(* Logix 5000 project; controller cal1632 1756-L62 rev 16.20; software revision 16.05; part 33 of 57 *)
(* tags used below, declared in another part *)
   FAULT : BOOL;
   HMI : BOOL;
   p01r03_lc3_ave_ctrl : CONTROL;
   p01r09_pb_global_reset : BOOL;
   p01r09_stretch_mode : BOOL;
   p02_real_from_hmi : hmi_real;
   p22_ai_amps : REAL;
   p22_ai_hz : REAL;
   p22_ai_speed : REAL;
   p22_ai_ts1_lc : REAL;
   p22_ao_selected_speed : REAL;
   p22_ao_torque : REAL;
   p22_ao_vfd : REAL;
   p22_control_word : INT;
   p22_dint_to_hmi : DINT[16];
   p22_do_close_nip_roll : BOOL;
   p22_real_to_hmi : REAL[112];
   p22_status_word : INT;
   p22_ts1_gear_ratio : REAL;
   p22_ts1_roll_diameter_ft : REAL;
   p22_vfd_input_max : REAL;
   p22_vfd_input_min : REAL;
   p22_vfd_output_max : REAL;
   p22_vfd_output_min : REAL;
   p22r03_vfd_out_scaling : SYS_SCP;
   p22r04 : routine;
   p22r04_speed_to_vfd_1 : SYS_SPEED_TO_VFD;
   p22r04_timer_fault : TIMER[4];
   p22r04_timer_warning : TIMER[4];
   p22r05 : routine;
   p22r05_timer_fault : TIMER[4];
   p22r05_timer_warning : TIMER[4];
   p22r06 : routine;
   p22r06_ave_lc : REAL;
   p22r06_lc_buffer : REAL[20];
   p22r06_lc_ctrl : CONTROL;
   p22r06_sample_timer : TIMER;
   p22r06_timer_fault : TIMER[4];
   p22r06_timer_warning : TIMER[4];
   p22r06_unload : DINT;
   p22r07 : routine;
   p22r07_timer_fault : TIMER[4];
   p22r07_timer_warning : TIMER[4];
   p22r09_mode_jog : BOOL;
   p22r09_mode_run : BOOL;
   p22r09_mode_thread : BOOL;
   p22r11 : routine;
(* P22_Tension_Stand_1, continued *)

ROUTINE R04_Output   (* ladder *)
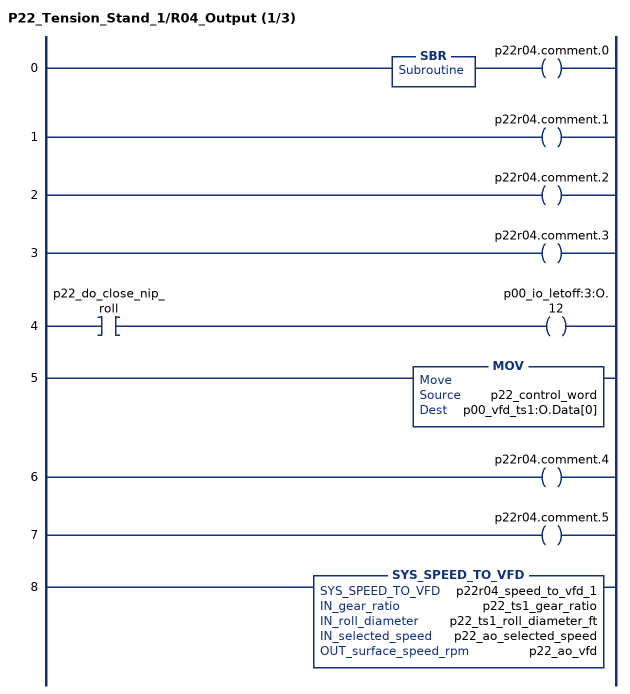
   0: SBR()OTE(p22r04.comment.0);
   1: OTE(p22r04.comment.1);
   2: OTE(p22r04.comment.2);
   3: OTE(p22r04.comment.3);
   4: XIC(p22_do_close_nip_roll)OTE(p00_io_letoff:3:O.12);
   5: MOV(p22_control_word,p00_vfd_ts1:O.Data[0]);
   6: OTE(p22r04.comment.4);
   7: OTE(p22r04.comment.5);
   8: SYS_SPEED_TO_VFD(p22r04_speed_to_vfd_1,p22_ts1_gear_ratio,p22_ts1_roll_diameter_ft,p22_ao_selected_speed,p22_ao_vfd);
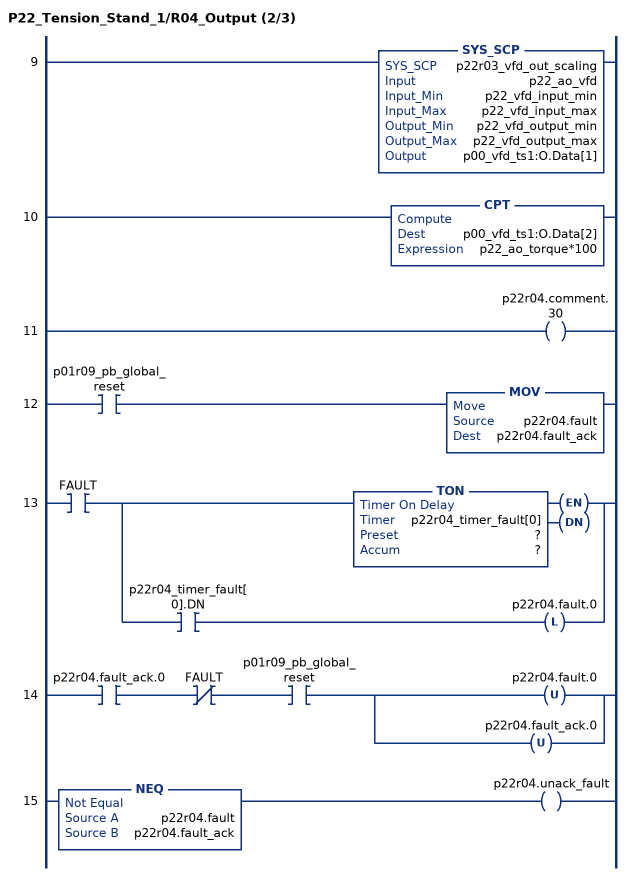
   9: SYS_SCP(p22r03_vfd_out_scaling,p22_ao_vfd,p22_vfd_input_min,p22_vfd_input_max,p22_vfd_output_min,p22_vfd_output_max,p00_vfd_ts1:O.Data[1]);
   10: CPT(p00_vfd_ts1:O.Data[2],p22_ao_torque*100);
   11: OTE(p22r04.comment.30);
   12: XIC(p01r09_pb_global_reset)MOV(p22r04.fault,p22r04.fault_ack);
   13: XIC(FAULT)[TON(p22r04_timer_fault[0],?,?) ,XIC(p22r04_timer_fault[0].DN) OTL(p22r04.fault.0) ];
   14: XIC(p22r04.fault_ack.0)XIO(FAULT)XIC(p01r09_pb_global_reset)[OTU(p22r04.fault.0) ,OTU(p22r04.fault_ack.0) ];
   15: NEQ(p22r04.fault,p22r04.fault_ack)OTE(p22r04.unack_fault);
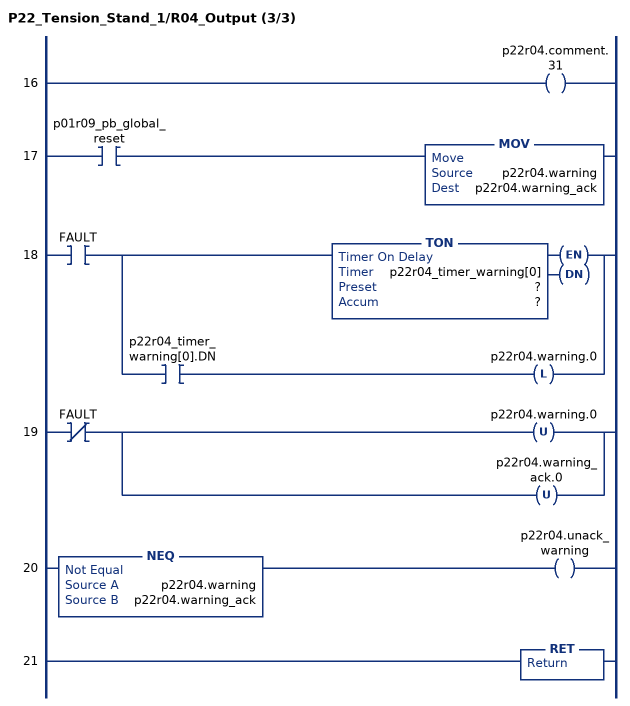
   16: OTE(p22r04.comment.31);
   17: XIC(p01r09_pb_global_reset)MOV(p22r04.warning,p22r04.warning_ack);
   18: XIC(FAULT)[TON(p22r04_timer_warning[0],?,?) ,XIC(p22r04_timer_warning[0].DN) OTL(p22r04.warning.0) ];
   19: XIO(FAULT)[OTU(p22r04.warning.0) ,OTU(p22r04.warning_ack.0) ];
   20: NEQ(p22r04.warning,p22r04.warning_ack)OTE(p22r04.unack_warning);
   21: RET();
END_ROUTINE

ROUTINE R05_Dint_to_HMI   (* ladder *)
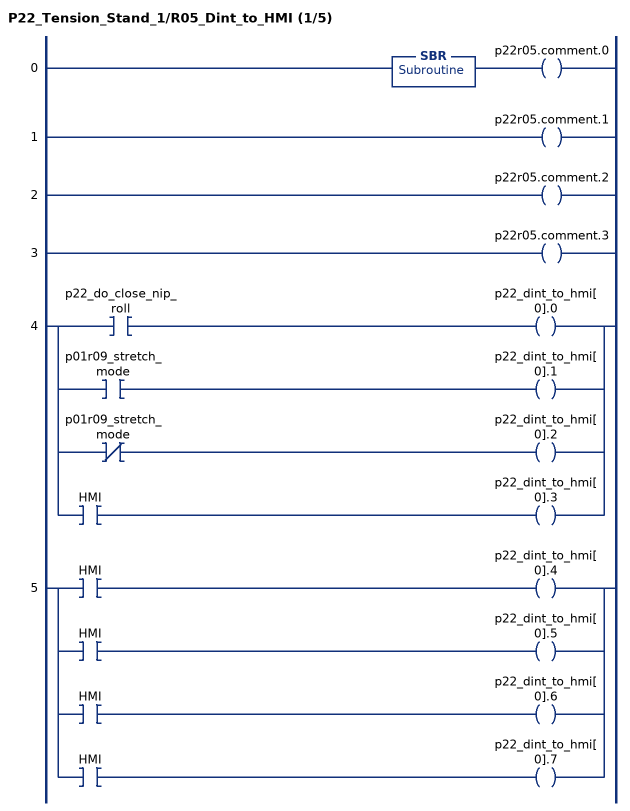
   0: SBR()OTE(p22r05.comment.0);
   1: OTE(p22r05.comment.1);
   2: OTE(p22r05.comment.2);
   3: OTE(p22r05.comment.3);
   4: [XIC(p22_do_close_nip_roll) OTE(p22_dint_to_hmi[0].0) ,XIC(p01r09_stretch_mode) OTE(p22_dint_to_hmi[0].1) ,XIO(p01r09_stretch_mode) OTE(p22_dint_to_hmi[0].2) ,XIC(HMI) OTE(p22_dint_to_hmi[0].3) ];
   5: [XIC(HMI) OTE(p22_dint_to_hmi[0].4) ,XIC(HMI) OTE(p22_dint_to_hmi[0].5) ,XIC(HMI) OTE(p22_dint_to_hmi[0].6) ,XIC(HMI) OTE(p22_dint_to_hmi[0].7) ];
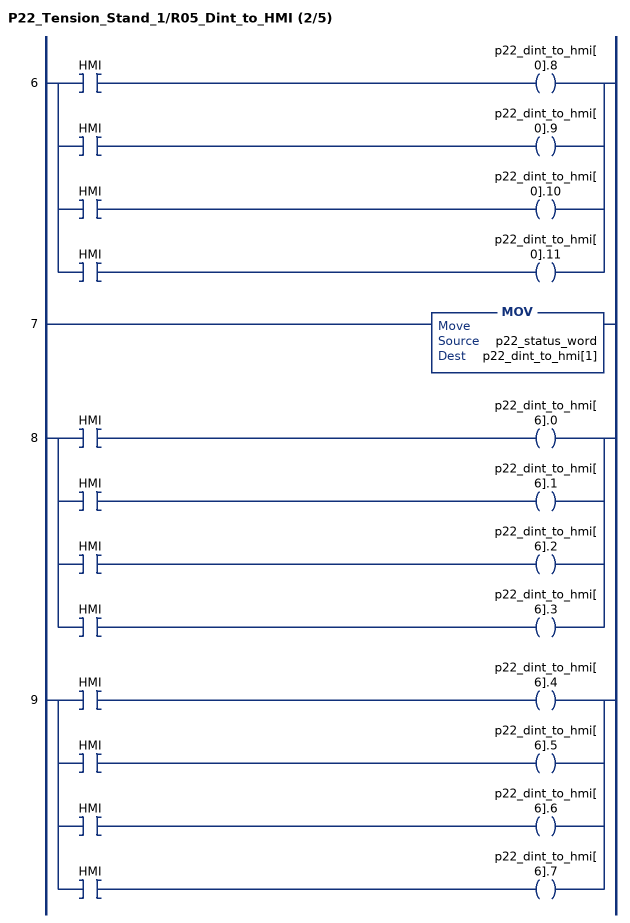
   6: [XIC(HMI) OTE(p22_dint_to_hmi[0].8) ,XIC(HMI) OTE(p22_dint_to_hmi[0].9) ,XIC(HMI) OTE(p22_dint_to_hmi[0].10) ,XIC(HMI) OTE(p22_dint_to_hmi[0].11) ];
   7: MOV(p22_status_word,p22_dint_to_hmi[1]);
   8: [XIC(HMI) OTE(p22_dint_to_hmi[6].0) ,XIC(HMI) OTE(p22_dint_to_hmi[6].1) ,XIC(HMI) OTE(p22_dint_to_hmi[6].2) ,XIC(HMI) OTE(p22_dint_to_hmi[6].3) ];
   9: [XIC(HMI) OTE(p22_dint_to_hmi[6].4) ,XIC(HMI) OTE(p22_dint_to_hmi[6].5) ,XIC(HMI) OTE(p22_dint_to_hmi[6].6) ,XIC(HMI) OTE(p22_dint_to_hmi[6].7) ];
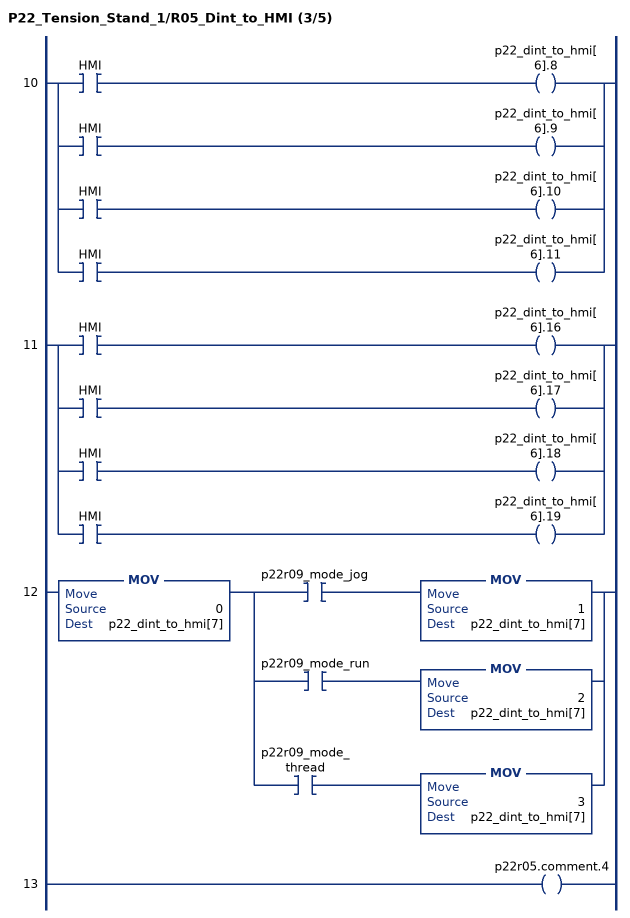
   10: [XIC(HMI) OTE(p22_dint_to_hmi[6].8) ,XIC(HMI) OTE(p22_dint_to_hmi[6].9) ,XIC(HMI) OTE(p22_dint_to_hmi[6].10) ,XIC(HMI) OTE(p22_dint_to_hmi[6].11) ];
   11: [XIC(HMI) OTE(p22_dint_to_hmi[6].16) ,XIC(HMI) OTE(p22_dint_to_hmi[6].17) ,XIC(HMI) OTE(p22_dint_to_hmi[6].18) ,XIC(HMI) OTE(p22_dint_to_hmi[6].19) ];
   12: MOV(0,p22_dint_to_hmi[7])[XIC(p22r09_mode_jog) MOV(1,p22_dint_to_hmi[7]) ,XIC(p22r09_mode_run) MOV(2,p22_dint_to_hmi[7]) ,XIC(p22r09_mode_thread) MOV(3,p22_dint_to_hmi[7]) ];
   13: OTE(p22r05.comment.4);
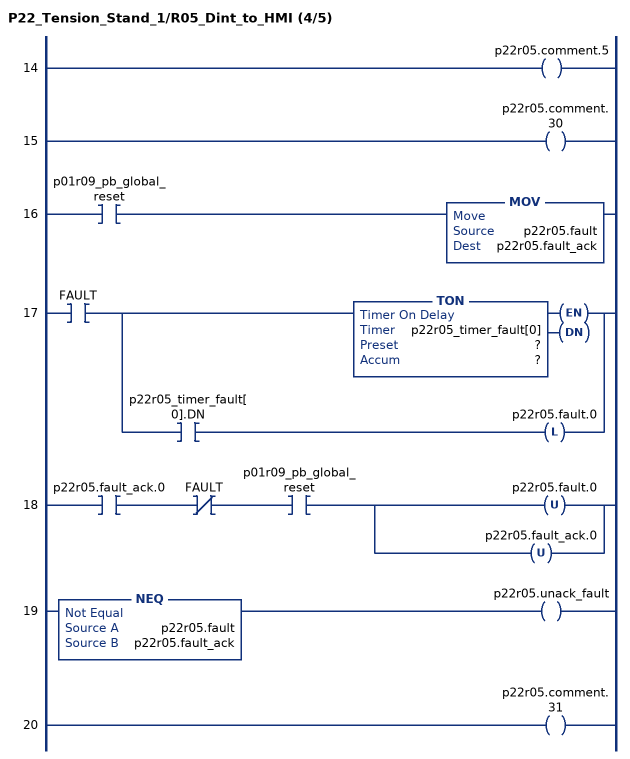
   14: OTE(p22r05.comment.5);
   15: OTE(p22r05.comment.30);
   16: XIC(p01r09_pb_global_reset)MOV(p22r05.fault,p22r05.fault_ack);
   17: XIC(FAULT)[TON(p22r05_timer_fault[0],?,?) ,XIC(p22r05_timer_fault[0].DN) OTL(p22r05.fault.0) ];
   18: XIC(p22r05.fault_ack.0)XIO(FAULT)XIC(p01r09_pb_global_reset)[OTU(p22r05.fault.0) ,OTU(p22r05.fault_ack.0) ];
   19: NEQ(p22r05.fault,p22r05.fault_ack)OTE(p22r05.unack_fault);
   20: OTE(p22r05.comment.31);
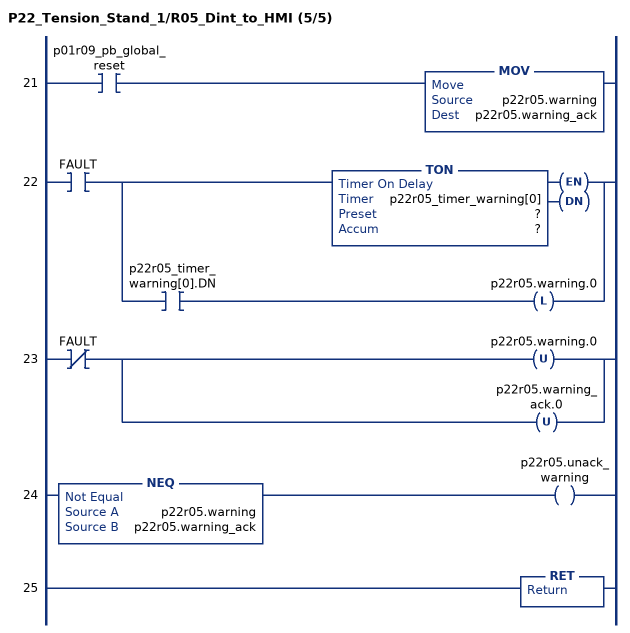
   21: XIC(p01r09_pb_global_reset)MOV(p22r05.warning,p22r05.warning_ack);
   22: XIC(FAULT)[TON(p22r05_timer_warning[0],?,?) ,XIC(p22r05_timer_warning[0].DN) OTL(p22r05.warning.0) ];
   23: XIO(FAULT)[OTU(p22r05.warning.0) ,OTU(p22r05.warning_ack.0) ];
   24: NEQ(p22r05.warning,p22r05.warning_ack)OTE(p22r05.unack_warning);
   25: RET();
END_ROUTINE

ROUTINE R06_Real_to_HMI   (* ladder *)
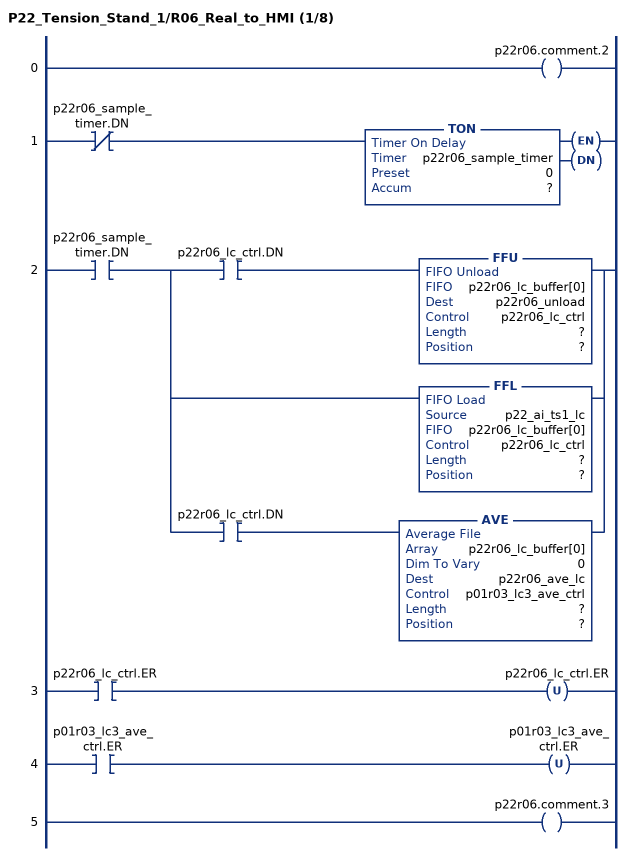
   0: OTE(p22r06.comment.2);
   1: XIO(p22r06_sample_timer.DN)TON(p22r06_sample_timer,?,?);
   2: XIC(p22r06_sample_timer.DN)[XIC(p22r06_lc_ctrl.DN) FFU(p22r06_lc_buffer[0],p22r06_unload,p22r06_lc_ctrl,?,?) ,FFL(p22_ai_ts1_lc,p22r06_lc_buffer[0],p22r06_lc_ctrl,?,?) ,XIC(p22r06_lc_ctrl.DN) AVE(p22r06_lc_buffer[0],0,p22r06_ave_lc,p01r03_lc3_ave_ctrl,?,?) ];
   3: XIC(p22r06_lc_ctrl.ER)OTU(p22r06_lc_ctrl.ER);
   4: XIC(p01r03_lc3_ave_ctrl.ER)OTU(p01r03_lc3_ave_ctrl.ER);
   5: OTE(p22r06.comment.3);
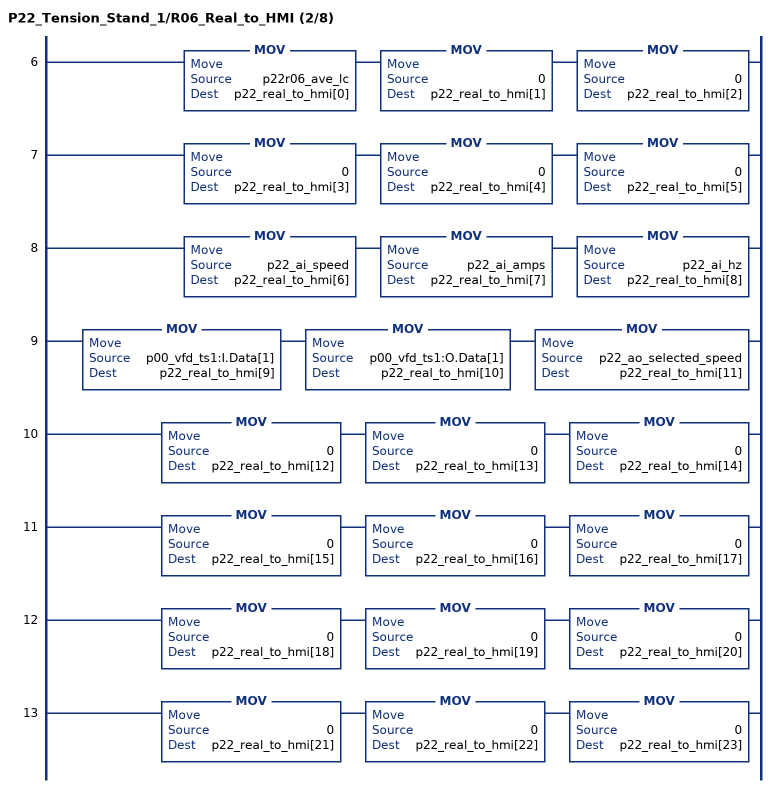
   6: MOV(p22r06_ave_lc,p22_real_to_hmi[0])MOV(0,p22_real_to_hmi[1])MOV(0,p22_real_to_hmi[2]);
   7: MOV(0,p22_real_to_hmi[3])MOV(0,p22_real_to_hmi[4])MOV(0,p22_real_to_hmi[5]);
   8: MOV(p22_ai_speed,p22_real_to_hmi[6])MOV(p22_ai_amps,p22_real_to_hmi[7])MOV(p22_ai_hz,p22_real_to_hmi[8]);
   9: MOV(p00_vfd_ts1:I.Data[1],p22_real_to_hmi[9])MOV(p00_vfd_ts1:O.Data[1],p22_real_to_hmi[10])MOV(p22_ao_selected_speed,p22_real_to_hmi[11]);
   10: MOV(0,p22_real_to_hmi[12])MOV(0,p22_real_to_hmi[13])MOV(0,p22_real_to_hmi[14]);
   11: MOV(0,p22_real_to_hmi[15])MOV(0,p22_real_to_hmi[16])MOV(0,p22_real_to_hmi[17]);
   12: MOV(0,p22_real_to_hmi[18])MOV(0,p22_real_to_hmi[19])MOV(0,p22_real_to_hmi[20]);
   13: MOV(0,p22_real_to_hmi[21])MOV(0,p22_real_to_hmi[22])MOV(0,p22_real_to_hmi[23]);
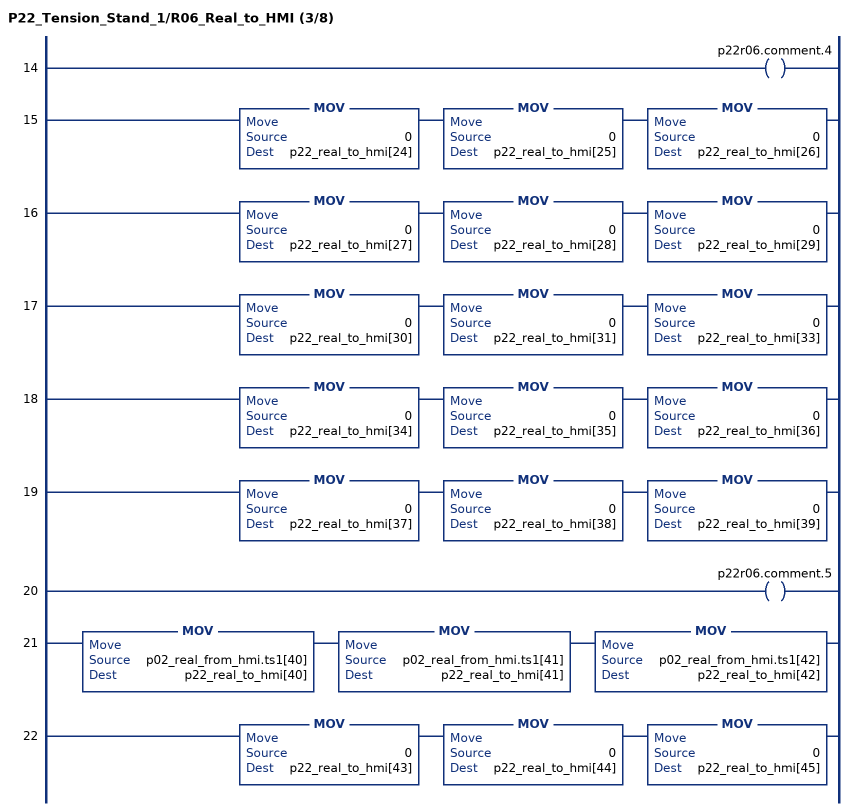
   14: OTE(p22r06.comment.4);
   15: MOV(0,p22_real_to_hmi[24])MOV(0,p22_real_to_hmi[25])MOV(0,p22_real_to_hmi[26]);
   16: MOV(0,p22_real_to_hmi[27])MOV(0,p22_real_to_hmi[28])MOV(0,p22_real_to_hmi[29]);
   17: MOV(0,p22_real_to_hmi[30])MOV(0,p22_real_to_hmi[31])MOV(0,p22_real_to_hmi[33]);
   18: MOV(0,p22_real_to_hmi[34])MOV(0,p22_real_to_hmi[35])MOV(0,p22_real_to_hmi[36]);
   19: MOV(0,p22_real_to_hmi[37])MOV(0,p22_real_to_hmi[38])MOV(0,p22_real_to_hmi[39]);
   20: OTE(p22r06.comment.5);
   21: MOV(p02_real_from_hmi.ts1[40],p22_real_to_hmi[40])MOV(p02_real_from_hmi.ts1[41],p22_real_to_hmi[41])MOV(p02_real_from_hmi.ts1[42],p22_real_to_hmi[42]);
   22: MOV(0,p22_real_to_hmi[43])MOV(0,p22_real_to_hmi[44])MOV(0,p22_real_to_hmi[45]);
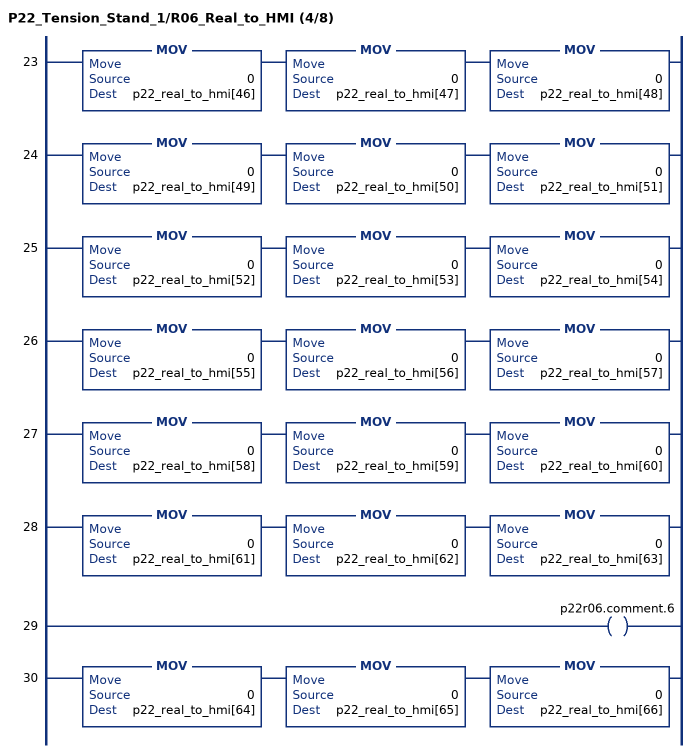
   23: MOV(0,p22_real_to_hmi[46])MOV(0,p22_real_to_hmi[47])MOV(0,p22_real_to_hmi[48]);
   24: MOV(0,p22_real_to_hmi[49])MOV(0,p22_real_to_hmi[50])MOV(0,p22_real_to_hmi[51]);
   25: MOV(0,p22_real_to_hmi[52])MOV(0,p22_real_to_hmi[53])MOV(0,p22_real_to_hmi[54]);
   26: MOV(0,p22_real_to_hmi[55])MOV(0,p22_real_to_hmi[56])MOV(0,p22_real_to_hmi[57]);
   27: MOV(0,p22_real_to_hmi[58])MOV(0,p22_real_to_hmi[59])MOV(0,p22_real_to_hmi[60]);
   28: MOV(0,p22_real_to_hmi[61])MOV(0,p22_real_to_hmi[62])MOV(0,p22_real_to_hmi[63]);
   29: OTE(p22r06.comment.6);
   30: MOV(0,p22_real_to_hmi[64])MOV(0,p22_real_to_hmi[65])MOV(0,p22_real_to_hmi[66]);
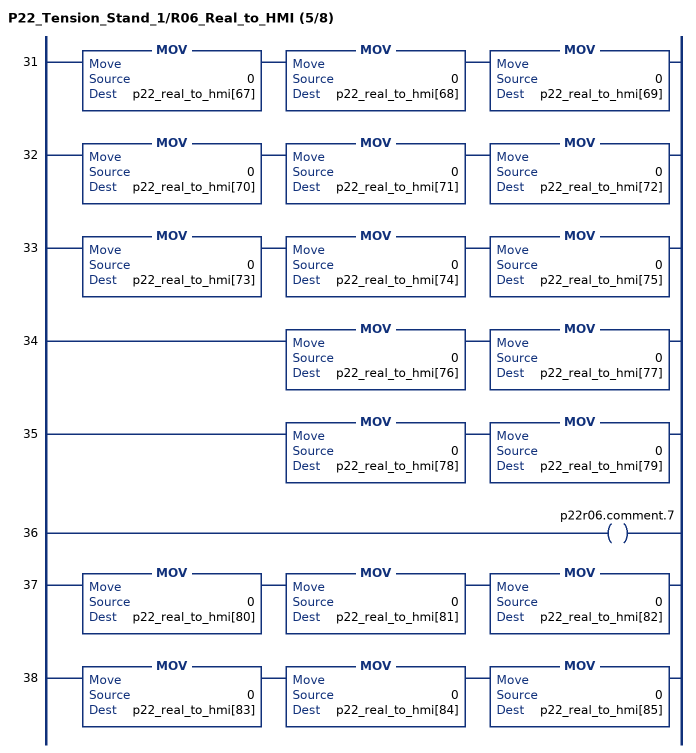
   31: MOV(0,p22_real_to_hmi[67])MOV(0,p22_real_to_hmi[68])MOV(0,p22_real_to_hmi[69]);
   32: MOV(0,p22_real_to_hmi[70])MOV(0,p22_real_to_hmi[71])MOV(0,p22_real_to_hmi[72]);
   33: MOV(0,p22_real_to_hmi[73])MOV(0,p22_real_to_hmi[74])MOV(0,p22_real_to_hmi[75]);
   34: MOV(0,p22_real_to_hmi[76])MOV(0,p22_real_to_hmi[77]);
   35: MOV(0,p22_real_to_hmi[78])MOV(0,p22_real_to_hmi[79]);
   36: OTE(p22r06.comment.7);
   37: MOV(0,p22_real_to_hmi[80])MOV(0,p22_real_to_hmi[81])MOV(0,p22_real_to_hmi[82]);
   38: MOV(0,p22_real_to_hmi[83])MOV(0,p22_real_to_hmi[84])MOV(0,p22_real_to_hmi[85]);
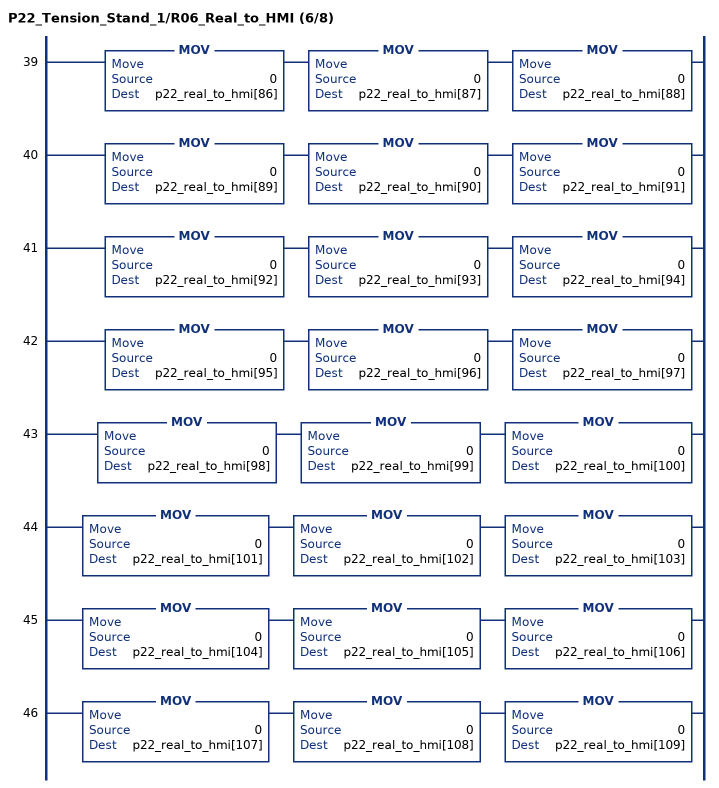
   39: MOV(0,p22_real_to_hmi[86])MOV(0,p22_real_to_hmi[87])MOV(0,p22_real_to_hmi[88]);
   40: MOV(0,p22_real_to_hmi[89])MOV(0,p22_real_to_hmi[90])MOV(0,p22_real_to_hmi[91]);
   41: MOV(0,p22_real_to_hmi[92])MOV(0,p22_real_to_hmi[93])MOV(0,p22_real_to_hmi[94]);
   42: MOV(0,p22_real_to_hmi[95])MOV(0,p22_real_to_hmi[96])MOV(0,p22_real_to_hmi[97]);
   43: MOV(0,p22_real_to_hmi[98])MOV(0,p22_real_to_hmi[99])MOV(0,p22_real_to_hmi[100]);
   44: MOV(0,p22_real_to_hmi[101])MOV(0,p22_real_to_hmi[102])MOV(0,p22_real_to_hmi[103]);
   45: MOV(0,p22_real_to_hmi[104])MOV(0,p22_real_to_hmi[105])MOV(0,p22_real_to_hmi[106]);
   46: MOV(0,p22_real_to_hmi[107])MOV(0,p22_real_to_hmi[108])MOV(0,p22_real_to_hmi[109]);
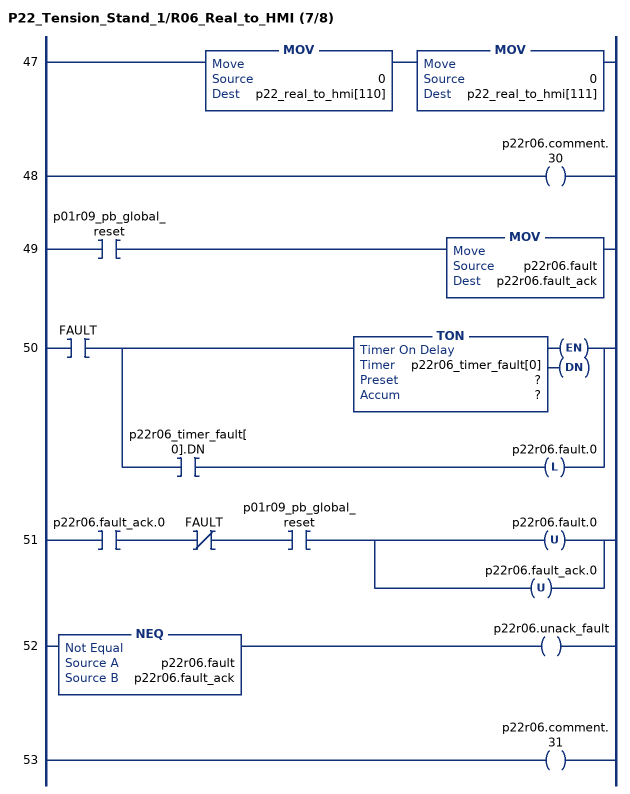
   47: MOV(0,p22_real_to_hmi[110])MOV(0,p22_real_to_hmi[111]);
   48: OTE(p22r06.comment.30);
   49: XIC(p01r09_pb_global_reset)MOV(p22r06.fault,p22r06.fault_ack);
   50: XIC(FAULT)[TON(p22r06_timer_fault[0],?,?) ,XIC(p22r06_timer_fault[0].DN) OTL(p22r06.fault.0) ];
   51: XIC(p22r06.fault_ack.0)XIO(FAULT)XIC(p01r09_pb_global_reset)[OTU(p22r06.fault.0) ,OTU(p22r06.fault_ack.0) ];
   52: NEQ(p22r06.fault,p22r06.fault_ack)OTE(p22r06.unack_fault);
   53: OTE(p22r06.comment.31);
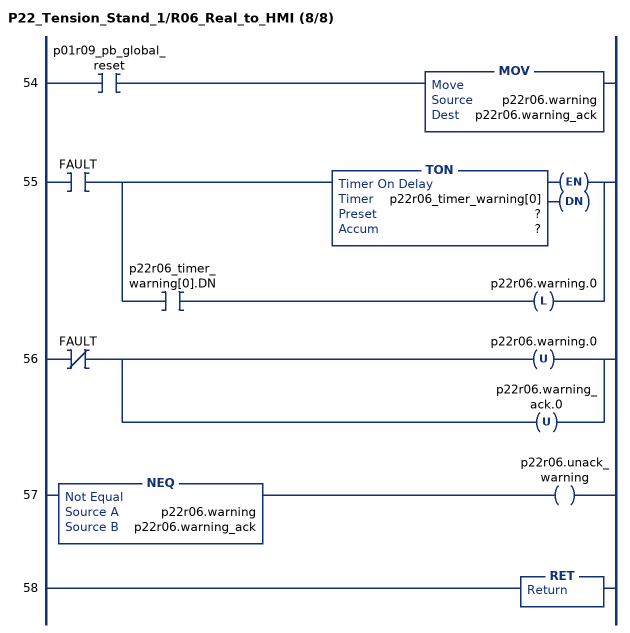
   54: XIC(p01r09_pb_global_reset)MOV(p22r06.warning,p22r06.warning_ack);
   55: XIC(FAULT)[TON(p22r06_timer_warning[0],?,?) ,XIC(p22r06_timer_warning[0].DN) OTL(p22r06.warning.0) ];
   56: XIO(FAULT)[OTU(p22r06.warning.0) ,OTU(p22r06.warning_ack.0) ];
   57: NEQ(p22r06.warning,p22r06.warning_ack)OTE(p22r06.unack_warning);
   58: RET();
END_ROUTINE

ROUTINE R07_Alarms   (* ladder *)
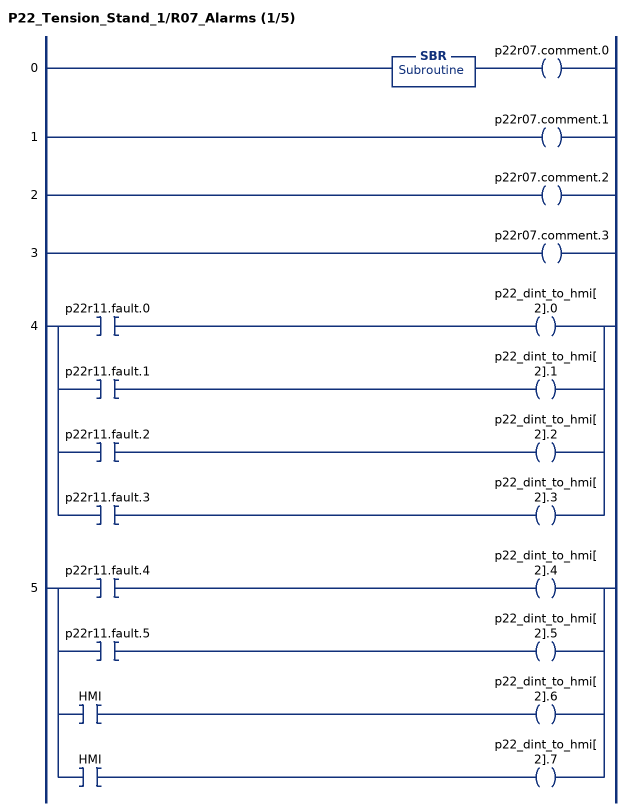
   0: SBR()OTE(p22r07.comment.0);
   1: OTE(p22r07.comment.1);
   2: OTE(p22r07.comment.2);
   3: OTE(p22r07.comment.3);
   4: [XIC(p22r11.fault.0) OTE(p22_dint_to_hmi[2].0) ,XIC(p22r11.fault.1) OTE(p22_dint_to_hmi[2].1) ,XIC(p22r11.fault.2) OTE(p22_dint_to_hmi[2].2) ,XIC(p22r11.fault.3) OTE(p22_dint_to_hmi[2].3) ];
   5: [XIC(p22r11.fault.4) OTE(p22_dint_to_hmi[2].4) ,XIC(p22r11.fault.5) OTE(p22_dint_to_hmi[2].5) ,XIC(HMI) OTE(p22_dint_to_hmi[2].6) ,XIC(HMI) OTE(p22_dint_to_hmi[2].7) ];
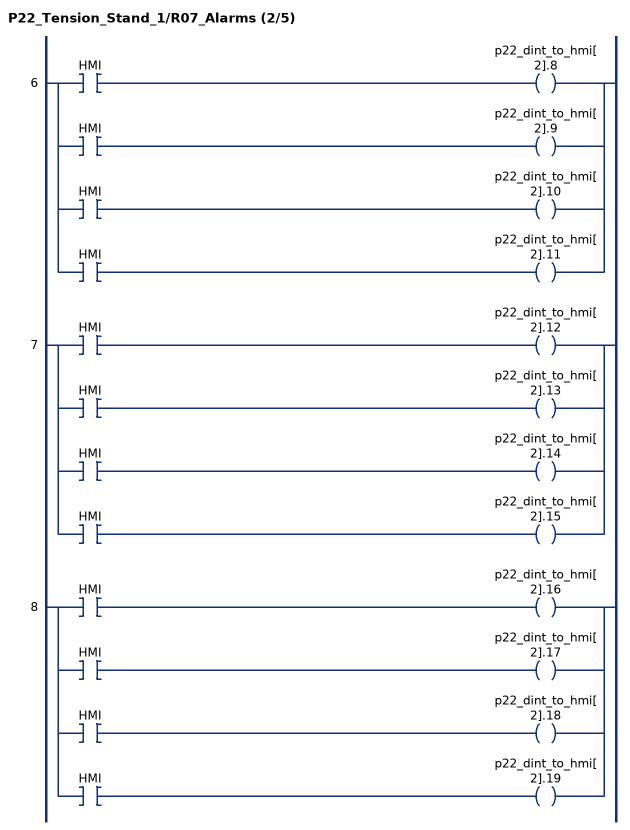
   6: [XIC(HMI) OTE(p22_dint_to_hmi[2].8) ,XIC(HMI) OTE(p22_dint_to_hmi[2].9) ,XIC(HMI) OTE(p22_dint_to_hmi[2].10) ,XIC(HMI) OTE(p22_dint_to_hmi[2].11) ];
   7: [XIC(HMI) OTE(p22_dint_to_hmi[2].12) ,XIC(HMI) OTE(p22_dint_to_hmi[2].13) ,XIC(HMI) OTE(p22_dint_to_hmi[2].14) ,XIC(HMI) OTE(p22_dint_to_hmi[2].15) ];
   8: [XIC(HMI) OTE(p22_dint_to_hmi[2].16) ,XIC(HMI) OTE(p22_dint_to_hmi[2].17) ,XIC(HMI) OTE(p22_dint_to_hmi[2].18) ,XIC(HMI) OTE(p22_dint_to_hmi[2].19) ];
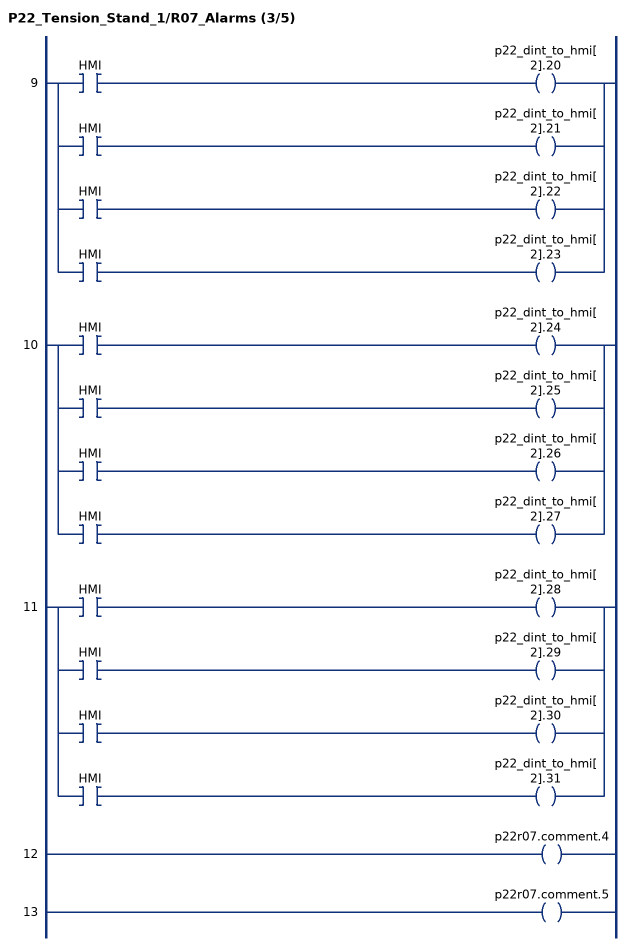
   9: [XIC(HMI) OTE(p22_dint_to_hmi[2].20) ,XIC(HMI) OTE(p22_dint_to_hmi[2].21) ,XIC(HMI) OTE(p22_dint_to_hmi[2].22) ,XIC(HMI) OTE(p22_dint_to_hmi[2].23) ];
   10: [XIC(HMI) OTE(p22_dint_to_hmi[2].24) ,XIC(HMI) OTE(p22_dint_to_hmi[2].25) ,XIC(HMI) OTE(p22_dint_to_hmi[2].26) ,XIC(HMI) OTE(p22_dint_to_hmi[2].27) ];
   11: [XIC(HMI) OTE(p22_dint_to_hmi[2].28) ,XIC(HMI) OTE(p22_dint_to_hmi[2].29) ,XIC(HMI) OTE(p22_dint_to_hmi[2].30) ,XIC(HMI) OTE(p22_dint_to_hmi[2].31) ];
   12: OTE(p22r07.comment.4);
   13: OTE(p22r07.comment.5);
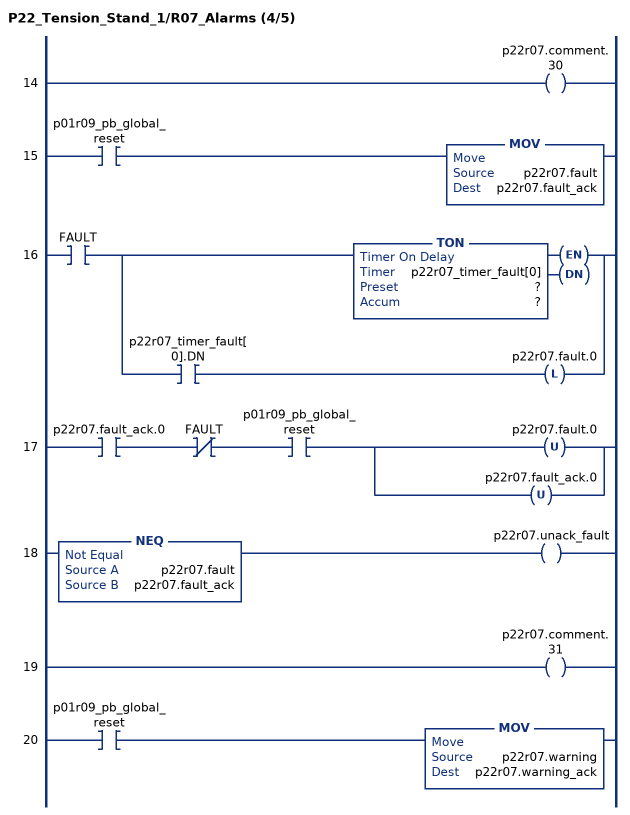
   14: OTE(p22r07.comment.30);
   15: XIC(p01r09_pb_global_reset)MOV(p22r07.fault,p22r07.fault_ack);
   16: XIC(FAULT)[TON(p22r07_timer_fault[0],?,?) ,XIC(p22r07_timer_fault[0].DN) OTL(p22r07.fault.0) ];
   17: XIC(p22r07.fault_ack.0)XIO(FAULT)XIC(p01r09_pb_global_reset)[OTU(p22r07.fault.0) ,OTU(p22r07.fault_ack.0) ];
   18: NEQ(p22r07.fault,p22r07.fault_ack)OTE(p22r07.unack_fault);
   19: OTE(p22r07.comment.31);
   20: XIC(p01r09_pb_global_reset)MOV(p22r07.warning,p22r07.warning_ack);
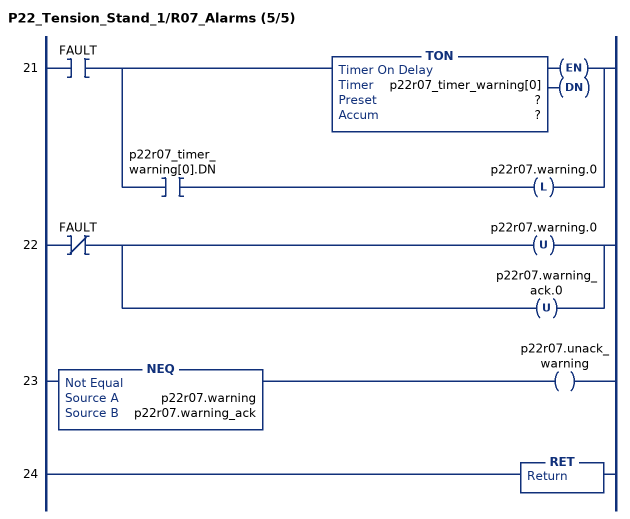
   21: XIC(FAULT)[TON(p22r07_timer_warning[0],?,?) ,XIC(p22r07_timer_warning[0].DN) OTL(p22r07.warning.0) ];
   22: XIO(FAULT)[OTU(p22r07.warning.0) ,OTU(p22r07.warning_ack.0) ];
   23: NEQ(p22r07.warning,p22r07.warning_ack)OTE(p22r07.unack_warning);
   24: RET();
END_ROUTINE
